TYPE (* logiBUS DI Events Struct Dual *)
  (* Version 1.0, 2026-05-28, franz *)
  PACKAGE logiBUS::io::DI;
  IMPORT eclipse4diac::core::TypeHash;
  IMPORT logiBUS::io::DI::logiBUS_DI_Events_S;
  logiBUS_DI_Events_S_Dual : STRUCT
    Up : logiBUS::io::DI::logiBUS_DI_Events_S; (* forward, up, right, clockwise *)
    Down : logiBUS::io::DI::logiBUS_DI_Events_S; (* backward, down, left, counter-clockwise *)
  END_STRUCT;
END_TYPE
